IF (TRIG_valve_tank_R.Q	OR Timer_valveQ = TRUE) THEN
	HW_valve_pomp_teplica :=	FALSE;
	Timer_valveQ	:= FALSE;
	Timer_valve.IN	:= FALSE;
END_IF



IF (TRIG_start_poliv.Q AND  Modbus.Teplica_poliv_status_PLC <> 2)   THEN
		Cnt_cleared	:= 	FALSE;
		Step_1_clear	 :=	FALSE;
		Poliv_liters	:=	0;
		FertA_liters	:=	0;
		FertB_liters	:=	0;
		Cnt_water_fertA_start	:=	0;
		Cnt_water_fertB_start	:=	0;
		Modbus.Cnt_water_fertA	:=	0;
		Modbus.Cnt_water_fertB	:=	0;
		Modbus.Teplica_DI1_poliv	:=	0;
		Modbus.Teplica_DI2_fertA	:=	0;
		Modbus.Teplica_DI3_fertB	:=	0;
		Modbus.Teplica_poliv_status_PLC:=1;
		Modbus.Teplica_poliv_message_PLC:=1;
		Modbus.Teplica_time_elapsed_poliv :=0;
		Modbus.Teplica_time_elapsed_fertA :=0;
		Modbus.Teplica_time_elapsed_fertB :=0;

		Timer_1_clearQ			:= FALSE;
		Timer_2_fertAQ			:= FALSE;
		Timer_3_clearQ			:= FALSE;
		Timer_4_fertBQ			:= FALSE;
		Step_1_clear				:= FALSE;
		Poliv_init_stop			:= FALSE;
		FertA_init_stop			:=	FALSE;
		FertB_init_stop			:=	FALSE;
		Bool_poliv_before_fert		:=	FALSE;
END_IF

(*ограничитель полива  в случае невозможности обнулить счётчики из-за недоступности RS485-шлюза*)
(*
	IF (Poliv_init_stop	=	FALSE AND (Modbus.Teplica_poliv_break=TRUE  OR  Cnt_Teplica_poliv_message_PLC_M3 > 2 OR  Cnt_Teplica_poliv_message_PLC_M5 > 2 OR  Cnt_Teplica_poliv_message_PLC_M7 > 2 OR  Cnt_Teplica_poliv_message_PLC_M9 > 2 OR  Cnt_Teplica_poliv_message_PLC_M11 > 2))
	THEN
		Cnt_cleared	:= 	FALSE;
		Modbus.Teplica_poliv_status_PLC :=  0;
		Poliv_init_stop	:=	TRUE;
		Modbus.Teplica_poliv_active:= FALSE;

		Modbus.Teplica_DO4_pomp_poliv:=FALSE;
		Modbus.Teplica_DO5_pomp_fertA :=  FALSE;
		Modbus.Teplica_DO6_pomp_fertB :=  FALSE;

		Step_1_clear	 :=	FALSE;

		Timer_poliv_all.IN := FALSE;
		Timer_1_clear.IN := FALSE;
		Timer_2_fertA.IN:=FALSE;
		Timer_3_clear.IN := FALSE;
		Timer_4_fertB.IN:=FALSE;
	END_IF
*)

(*Нормальный режим старта полива после обнуления счётчиков*)

IF (Modbus.Teplica_poliv_status_PLC=2 AND Cnt_cleared=TRUE AND Step_1_clear = FALSE ) THEN
	DO3_poliv_writed_0		:=	FALSE;
	DO4_fertA_writed_0		:=	FALSE;
	DO5_fertB_writed_0		:=	FALSE;

	Step_1_clear	 :=	TRUE;
	Modbus.Teplica_DO4_pomp_poliv:=TRUE;
	 t_Started_poliv := TIME();
	Timer_poliv_all(IN:=NOT Timer_poliv_allQ , PT:=tTimerValue_poliv_all , Q=>Timer_poliv_allQ , ET=> );
	Timer_poliv_with_fert(IN:=NOT Timer_poliv_with_fertQ , PT:=tTimerValue_poliv_with_fert , Q=>Timer_poliv_with_fertQ , ET=> );
	Timer_1_clear(IN:=NOT Timer_1_clearQ , PT:=tTimerValue_1_clear , Q=>Timer_1_clearQ , ET=> );
END_IF

IF (Modbus.Teplica_poliv_status_PLC=2 AND Cnt_cleared=TRUE  ) THEN


	Poliv_liters 	:= 	UDINT_TO_REAL(Modbus.Teplica_DI1_poliv)/INT_TO_REAL(Modbus.Teplica_poliv_kf);
	FertA_liters	:=	UDINT_TO_REAL(Modbus.Teplica_DI2_fertA)/INT_TO_REAL(Modbus.Teplica_fertA_kf);
	FertB_liters	:=	UDINT_TO_REAL(Modbus.Teplica_DI3_fertB)/INT_TO_REAL(Modbus.Teplica_fertB_kf);
	Modbus.Teplica_time_elapsed_poliv :=(TIME_TO_UDINT( TIME() - t_Started_poliv))/1000;

(* промывка и фертигация   OR Modbus.Teplica_set_poliv_before_fert >Poliv_liters*)

IF (Modbus.Teplica_type_poliv = TRUE) THEN
	IF ((Timer_1_clear.Q OR Poliv_liters>Modbus.Teplica_set_poliv_before_fert) AND Bool_poliv_before_fert=FALSE) THEN
		Timer_1_clear.IN 		:= FALSE;
		Bool_poliv_before_fert	:= TRUE;
		IF (Modbus.Teplica_type_fert = FALSE) THEN
			Modbus.Teplica_DO5_pomp_fertA :=  TRUE;  (*включение насоса фертигации из бака А*)
			Timer_2_fertA(IN:=NOT Timer_2_fertAQ , PT:=tTimerValue_2_fertA , Q=>Timer_2_fertAQ , ET=> );
			t_Started_fertA := TIME();
			Cnt_water_fertA_start :=Modbus.Teplica_DI1_poliv;


		ELSE
			Modbus.Teplica_DO6_pomp_fertB :=  TRUE;   (*включение насоса фертигации из бака B*)
			Timer_4_fertB(IN:=NOT Timer_4_fertBQ , PT:=tTimerValue_4_fertB , Q=>Timer_4_fertBQ , ET=> );
			t_Started_fertB := TIME();
			Cnt_water_fertB_start :=Modbus.Teplica_DI1_poliv;

		END_IF


	END_IF





	IF ( (Timer_2_fertA.Q OR FertA_liters > Modbus.Teplica_set_fertA) AND Modbus.Teplica_DO5_pomp_fertA =  TRUE) THEN
		Modbus.Teplica_DO5_pomp_fertA :=  FALSE; (*отключение насоса фертигации из бака А*)
		Timer_2_fertA.IN:=FALSE;
		FertA_init_stop	:=	TRUE;
		Timer_3_clear(IN:=NOT Timer_3_clearQ , PT:=tTimerValue_3_clear , Q=>Timer_3_clearQ , ET=> );
	END_IF

	IF ( (Timer_4_fertB.Q OR FertB_liters > Modbus.Teplica_set_fertB) AND Modbus.Teplica_DO6_pomp_fertB =  TRUE ) THEN
		Modbus.Teplica_DO6_pomp_fertB :=  FALSE; (*отключение насоса фертигации из бака B*)
		Timer_4_fertB.IN:=FALSE;
		FertB_init_stop	:=	TRUE;
		Timer_3_clear(IN:=NOT Timer_3_clearQ , PT:=tTimerValue_3_clear , Q=>Timer_3_clearQ , ET=> );
	END_IF

END_IF

(*ограничитель полива  в нормальном режиме*)
	IF (Modbus.Teplica_type_poliv = FALSE) THEN
		IF ((Timer_poliv_all.Q=TRUE OR (Poliv_liters > Modbus.Teplica_set_poliv)  OR Modbus.Teplica_poliv_break=TRUE OR Timer_3_clear.Q=TRUE) AND  Poliv_init_stop = FALSE )THEN
			IF (Modbus.Teplica_DO5_pomp_fertA =  TRUE) THEN
				Modbus.Teplica_time_elapsed_fertA :=(TIME_TO_UDINT( TIME() - t_Started_fertA))/1000;
			END_IF
			IF (Modbus.Teplica_DO6_pomp_fertB =  TRUE) THEN
				Modbus.Teplica_time_elapsed_fertB :=(TIME_TO_UDINT( TIME() - t_Started_fertB))/1000;
			END_IF

			Poliv_init_stop	:=	TRUE;
			Cnt_cleared	:= 	FALSE;
			Modbus.Teplica_poliv_status_PLC :=  0;
			Modbus.Teplica_poliv_active:= FALSE;
			Modbus.Teplica_DO4_pomp_poliv:=FALSE;
			Modbus.Teplica_DO5_pomp_fertA :=  FALSE;
			Modbus.Teplica_DO6_pomp_fertB :=  FALSE;
			Timer_poliv_all.IN := FALSE;
			Timer_poliv_with_fert.IN := FALSE;
			Timer_1_clear.IN := FALSE;
			Timer_2_fertA.IN:=FALSE;
			Timer_3_clear.IN := FALSE;
			Timer_4_fertB.IN:=FALSE;
		END_IF
	ELSE
		IF ((Timer_poliv_with_fert.Q=TRUE OR   Modbus.Teplica_poliv_break=TRUE OR Timer_3_clear.Q=TRUE) AND  Poliv_init_stop = FALSE )THEN
			IF (Modbus.Teplica_DO5_pomp_fertA =  TRUE) THEN
				Modbus.Teplica_time_elapsed_fertA :=(TIME_TO_UDINT( TIME() - t_Started_fertA))/1000;
			END_IF
			IF (Modbus.Teplica_DO6_pomp_fertB =  TRUE) THEN
				Modbus.Teplica_time_elapsed_fertB :=(TIME_TO_UDINT( TIME() - t_Started_fertB))/1000;
			END_IF

			Poliv_init_stop	:=	TRUE;
			Cnt_cleared	:= 	FALSE;
			Modbus.Teplica_poliv_status_PLC :=  0;
			Modbus.Teplica_poliv_active:= FALSE;
			Modbus.Teplica_DO4_pomp_poliv:=FALSE;
			Modbus.Teplica_DO5_pomp_fertA :=  FALSE;
			Modbus.Teplica_DO6_pomp_fertB :=  FALSE;
			Timer_poliv_all.IN := FALSE;
			Timer_poliv_with_fert.IN := FALSE;
			Timer_1_clear.IN := FALSE;
			Timer_2_fertA.IN:=FALSE;
			Timer_3_clear.IN := FALSE;
			Timer_4_fertB.IN:=FALSE;
		END_IF
	END_IF
END_IF











(*LIGHT TEPLICA *)

IF (Modbus.Teplica_DO3_light = FALSE) THEN

	IF ((Modbus.Teplica_light_lux > Modbus.Teplica_light_set_low+gisterezis_lux) OR Modbus.Teplica_light_allow = FALSE  ) THEN
		Modbus.Teplica_DO3_light :=FALSE;
	END_IF

	IF ((Modbus.Teplica_light_lux <  Modbus.Teplica_light_set_low-gisterezis_lux ) AND Modbus.Teplica_light_allow ) THEN
		Modbus.Teplica_DO3_light:=TRUE;
	END_IF

END_IF

IF (Modbus.Teplica_DO3_light = TRUE) THEN

	IF ((Modbus.Teplica_light_lux-Modbus.Teplica_power_light_lux > Modbus.Teplica_light_set_low+gisterezis_lux) OR Modbus.Teplica_light_allow = FALSE  ) THEN
		Modbus.Teplica_DO3_light :=FALSE;
	END_IF

	IF ((Modbus.Teplica_light_lux-Modbus.Teplica_power_light_lux <  Modbus.Teplica_light_set_low-gisterezis_lux ) AND Modbus.Teplica_light_allow ) THEN
		Modbus.Teplica_DO3_light:=TRUE;
	END_IF

END_IF



(*HEAT TEPLICA *)

	IF ((Modbus.Teplica_temp_air > Modbus.Teplica_temp_set_low+1)   ) THEN
		Modbus.Teplica_DO2_heat :=FALSE;
	END_IF

	IF ((Modbus.Teplica_temp_air <  Modbus.Teplica_temp_set_low-1 ) ) THEN
		Modbus.Teplica_DO2_heat:=TRUE;
	END_IF

(*VENT  TEPLICA *)

	IF ((Modbus.Teplica_temp_air < Modbus.Teplica_temp_set_high-1)   ) THEN
		Modbus.Teplica_DO1_vent			 :=FALSE;
	END_IF

	IF ((Modbus.Teplica_temp_air >  Modbus.Teplica_temp_set_high+1 ) ) THEN
		Modbus.Teplica_DO1_vent:=TRUE;
	END_IF


	IF (Modbus.Teplica_temp_air < Modbus.Teplica_set_temp_window_open-1 ) THEN
		HW_window_opener				:=FALSE;
		Modbus.Teplica_window_opener	:=FALSE;
	END_IF
	IF (Modbus.Teplica_temp_air >  Modbus.Teplica_set_temp_window_open+1 AND   Modbus.Street_temp > 5 ) THEN
		HW_window_opener				:=TRUE;
		Modbus.Teplica_window_opener	:=TRUE;
	END_IF


	IF (Modbus.Teplica_temp_air < Modbus.Teplica_set_temp_pomp_cold-2   ) THEN
		HW_pomp_cold				:=FALSE;
		Modbus.Teplica_pomp_cold	:=FALSE;
	END_IF
	IF (Modbus.Teplica_temp_air >  Modbus.Teplica_set_temp_pomp_cold+2 AND   Modbus.Street_temp > 5 ) THEN
		HW_pomp_cold				:=TRUE;
		Modbus.Teplica_pomp_cold	:=TRUE;
	END_IF
END_PROGRAM

(* POU teplica_ai, ST *)
PROGRAM teplica_ai
VAR
    (* Общие таймеры *)
    Timer_poliv_all : TON;
    Timer_poliv_with_fert : TON;
    Timer_1_clear : TON;
    Timer_3_clear : TON;
    Timer_poliv_finish : TON;
    Timer_calc_kf : TON;
    Timer_valve : TON;

    (* Таймеры для баков (A и B) *)
    Timer_fert : ARRAY[1..2] OF TON;
    Timer_fertQ : ARRAY[1..2] OF BOOL;

    (* Триггеры *)
    TRIG_start_poliv : R_TRIG;
    TRIG_poliv_break : R_TRIG;
    TRIG_valve_tank_F : F_TRIG;
    TRIG_valve_tank_R : R_TRIG;
    TRIG_level_tank_low : R_TRIG;
    TRIG_level_tank_high : R_TRIG;

    (* ПИ-регуляторы и их параметры (для двух баков) *)
    pi_fert : ARRAY[1..2] OF FB_CTRL_PI;
    pi_par : ARRAY[1..2] OF ST_CTRL_PI_PARAMS;
    kf_calc : ARRAY[1..2] OF REAL;
    cnt_water_fert_start : ARRAY[1..2] OF UDINT;
    cnt_fert_calc_start : ARRAY[1..2] OF REAL;
    vol_fert : ARRAY[1..2] OF REAL;
    fOut : ARRAY[1..2] OF REAL;
    act : ARRAY[1..2] OF REAL;
    pwm_data : ARRAY[1..2] OF REAL;
    pwm_cnt : ARRAY[1..2] OF UDINT;
    pwm_avg : ARRAY[1..2] OF REAL;
    fert_pwm_level : ARRAY[1..2] OF UINT;

    (* Переменные для объёмов *)
    Poliv_liters : REAL;
    FertA_liters : REAL;
    FertB_liters : REAL;
    Cnt_water_calc_kf_start : REAL;
    vol_water : REAL;

    (* Прочие переменные *)
    Cnt_water_pipe : UDINT;
    Cnt_water_finish_clear_start : UDINT;
    Cnt_water_finish_clear : REAL;
    t_Started_poliv : TIME;
    t_Started_fert : ARRAY[1..2] OF TIME;
    tTimerValue_poliv_all : TIME := t#60s;
    tTimerValue_1_clear : TIME := t#10s;
    tTimerValue_2_fert : ARRAY[1..2] OF TIME := t#30s, t#10s;
    tTimerValue_3_clear : TIME := t#60s;
    tTimerValue_poliv_with_fert : TIME := t#60m;
    tTimerValue_poliv_finish : TIME := t#3s;
    tTimerValue_valve_water : TIME := t#60m;
    Bool_poliv_before_fert : BOOL;
    max_EC : REAL;
    avg_light_ma : FB_CTRL_MOVING_AVERAGE;
    stParams_avg_light : ST_CTRL_MOVING_AVERAGE_PARAMS;
    arr_table : ARRAY[1..20] OF FLOAT;
    start_cfg_avg_light : BOOL;
    start_cfg_pi_par : BOOL;
    gisterezis_lux : INT := 1000;
    tank_level_low : BOOL;
    tank_level_high : BOOL;
    fert_idx : INT;
    setpoint : REAL;
    zone_offset : INT;
END_VAR
(* ---------- Инициализация скользящего среднего ---------- *)
IF NOT start_cfg_avg_light THEN
    stParams_avg_light.tCtrlCycleTime := T#60s;
    stParams_avg_light.tTaskCycleTime := T#10ms;
    stParams_avg_light.nSamplesToFilter := 20;
    stParams_avg_light.pWorkArray_ADR := ADR(arr_table);
    stParams_avg_light.nWorkArray_SIZEOF := SIZEOF(arr_table);
    start_cfg_avg_light := TRUE;
END_IF
avg_light_ma(fIn:=Modbus.Teplica_light_lux, fManSyncValue:=0, bSync:=0,
             eMode:=eCTRL_MODE_ACTIVE, bHold:=0, stParams:=stParams_avg_light,
             fOut=>Modbus.Teplica_avg_lux);

(* ---------- Инициализация ПИ-регуляторов и коэффициентов ---------- *)
IF NOT start_cfg_pi_par THEN
    FOR fert_idx := 1 TO 2 DO
        pi_par[fert_idx].bARWOnIPartOnly := 0;
        pi_par[fert_idx].fKp := 300000;
        pi_par[fert_idx].fOutMaxLimit := 32765;
        pi_par[fert_idx].fOutMinLimit := 16800;
        pi_par[fert_idx].tCtrlCycleTime := T#4s;
        pi_par[fert_idx].tTaskCycleTime := T#10ms;
        pi_par[fert_idx].tTn := T#8s;
        kf_calc[fert_idx] := 12.0;   (* начальное значение Kf *)
    END_FOR
    start_cfg_pi_par := TRUE;
END_IF

(* ---------- Защита от нулевых коэффициентов ---------- *)
FOR fert_idx := 1 TO 2 DO
    IF kf_calc[fert_idx] = 0.0 THEN
        kf_calc[fert_idx] := 12.0;
    END_IF
END_FOR
IF Modbus.Teplica_fert_kf = 0 THEN
    Modbus.Teplica_fert_kf := 24;
END_IF
setpoint := 1.0 / INT_TO_REAL(Modbus.Teplica_fert_kf);

(* ---------- Установка времён из Modbus (перевод минут в мс) ---------- *)
tTimerValue_poliv_all        := UDINT_TO_TIME(60000 * Modbus.Teplica_set_max_poliv_time);
tTimerValue_1_clear          := UDINT_TO_TIME(60000 * Modbus.Teplica_set_clear_time);
tTimerValue_2_fert[1]        := UDINT_TO_TIME(60000 * Modbus.Teplica_set_max_fertA_time);
tTimerValue_2_fert[2]        := UDINT_TO_TIME(60000 * Modbus.Teplica_set_max_fertB_time);
tTimerValue_3_clear          := UDINT_TO_TIME(60000 * Modbus.Teplica_set_finish_clear_time);

(* ---------- Вызов таймеров ---------- *)
Timer_poliv_all();
Timer_poliv_with_fert();
Timer_1_clear();
Timer_3_clear();
FOR fert_idx := 1 TO 2 DO Timer_fert[fert_idx](); END_FOR
Timer_poliv_finish();
Timer_calc_kf();
Timer_valve();

(* ---------- Триггеры ---------- *)
TRIG_start_poliv(CLK := Modbus.Teplica_poliv_active);
TRIG_poliv_break(CLK := Modbus.Teplica_poliv_break);
TRIG_valve_tank_F(CLK := HW_water_tank_teplica_level);
TRIG_valve_tank_R(CLK := HW_water_tank_teplica_level);

tank_level_low   := Modbus.Teplica_tank_level < 1000;
tank_level_high  := Modbus.Teplica_tank_level > 1200;
TRIG_level_tank_low(CLK := tank_level_low);
TRIG_level_tank_high(CLK := tank_level_high);
Modbus.Teplica_tank_teplica_level := HW_water_tank_teplica_level;

(* ---------- Управление клапаном воды в бак ---------- *)
IF TRIG_valve_tank_F.Q OR TRIG_level_tank_low.Q THEN
    Timer_valve(IN := NOT Timer_valve.Q, PT := tTimerValue_valve_water);
    HW_valve_pomp_teplica := TRUE;
    Modbus.Teplica_valve_water_in := TRUE;
END_IF
IF TRIG_valve_tank_R.Q OR Timer_valve.Q OR TRIG_level_tank_high.Q THEN
    HW_valve_pomp_teplica := FALSE;
    Modbus.Teplica_valve_water_in := FALSE;
    Timer_valve.IN := FALSE;
END_IF

(* ---------- Старт полива ---------- *)
IF TRIG_start_poliv.Q AND Modbus.Teplica_tank_level > 400 THEN
    FOR fert_idx := 1 TO 2 DO
        pwm_data[fert_idx] := 0.0;
        pwm_cnt[fert_idx] := 0;
        pwm_avg[fert_idx] := 0.0;
        cnt_water_fert_start[fert_idx] := 0;
        cnt_fert_calc_start[fert_idx] := 0.0;
    END_FOR
    Modbus.Teplica_impulse_fertA_cnt := 0;
    Modbus.Teplica_impulse_fertB_cnt := 0;
    Modbus.Teplica_impulse_water_cnt := 0;
    Modbus.Teplica_cnt_water_pipe := 0;
    Modbus.Teplica_time_elapsed_poliv := 0;
    Modbus.Teplica_time_elapsed_fertA := 0;
    Modbus.Teplica_time_elapsed_fertB := 0;
    Poliv_liters := 0.0;
    FertA_liters := 0.0;
    FertB_liters := 0.0;
    Cnt_water_finish_clear := 0.0;
    Cnt_water_finish_clear_start := 0;
    Cnt_water_calc_kf_start := 0.0;
    max_EC := 0.0;
    Bool_poliv_before_fert := FALSE;

    FOR fert_idx := 1 TO 2 DO
        Timer_fert[fert_idx].IN := FALSE;
    END_FOR
    Timer_1_clear.IN := FALSE;
    Timer_3_clear.IN := FALSE;
    Timer_calc_kf.IN := FALSE;
    Timer_poliv_finish.IN := FALSE;
    Timer_poliv_all.IN := FALSE;
    Timer_poliv_with_fert.IN := FALSE;

    Modbus.Teplica_pomp_poliv := TRUE;
    t_Started_poliv := TIME();
    Timer_poliv_all(IN := NOT Timer_poliv_all.Q, PT := tTimerValue_poliv_all);
    Timer_poliv_with_fert(IN := NOT Timer_poliv_with_fert.Q, PT := tTimerValue_poliv_with_fert);
    Timer_1_clear(IN := NOT Timer_1_clear.Q, PT := tTimerValue_1_clear);
    Modbus.Teplica_poliv_status_PLC := 2;
    (* вычисляем смещение для зоны *)
    zone_offset := 0;
    IF Modbus.Teplica_zone_poliv <> 0 THEN zone_offset := 1; END_IF
    Modbus.Teplica_poliv_message_PLC := 1 + zone_offset;
END_IF

(* ---------- Основной цикл полива ---------- *)
IF Modbus.Teplica_poliv_status_PLC = 2 THEN
    Cnt_water_pipe := Modbus.Teplica_cnt_water_pipe;
    Poliv_liters  := UDINT_TO_REAL(Modbus.Teplica_impulse_water_cnt) / INT_TO_REAL(Modbus.Teplica_poliv_kf);
    FertA_liters  := UDINT_TO_REAL(Modbus.Teplica_impulse_fertA_cnt) / INT_TO_REAL(Modbus.Teplica_fertA_kf);
    FertB_liters  := UDINT_TO_REAL(Modbus.Teplica_impulse_fertB_cnt) / INT_TO_REAL(Modbus.Teplica_fertB_kf);
    Modbus.Teplica_time_elapsed_poliv := (TIME_TO_UDINT(TIME() - t_Started_poliv)) / 1000;
    IF Modbus.Teplica_sensor_soil_EC > max_EC THEN max_EC := Modbus.Teplica_sensor_soil_EC; END_IF

    (* выбор бака: 1 – A, 2 – B *)
    IF Modbus.Teplica_type_fert THEN
        fert_idx := 2;
    ELSE
        fert_idx := 1;
    END_IF

    (* смещение для зоны (используется далее) *)
    zone_offset := 0;
    IF Modbus.Teplica_zone_poliv <> 0 THEN zone_offset := 1; END_IF

    (* ------------------- Полив с фертигацией ------------------- *)
    IF Modbus.Teplica_type_poliv THEN
        (* Этап 1: промывка перед фертигацией *)
        IF NOT Timer_1_clear.Q AND NOT Bool_poliv_before_fert THEN
            Modbus.Teplica_poliv_message_PLC := 3 + (fert_idx-1)*2 + zone_offset;
        END_IF

        (* Переход к фертигации *)
        IF (Timer_1_clear.Q OR Poliv_liters > Modbus.Teplica_set_poliv_before_fert) AND NOT Bool_poliv_before_fert THEN
            Timer_1_clear.IN := FALSE;
            Bool_poliv_before_fert := TRUE;
            IF fert_idx = 1 THEN
                Modbus.Teplica_pomp_fertA := TRUE;
            ELSE
                Modbus.Teplica_pomp_fertB := TRUE;
            END_IF
            Timer_fert[fert_idx](IN := NOT Timer_fert[fert_idx].Q, PT := tTimerValue_2_fert[fert_idx]);
            t_Started_fert[fert_idx] := TIME();
            cnt_water_fert_start[fert_idx] := Modbus.Teplica_impulse_water_cnt;
            cnt_fert_calc_start[fert_idx] := Poliv_liters;
            Cnt_water_calc_kf_start := Poliv_liters;
            Modbus.Teplica_poliv_message_PLC := 7 + (fert_idx-1)*2 + zone_offset;
        END_IF

        (* Работа активного бака *)
        IF (fert_idx = 1 AND Modbus.Teplica_pomp_fertA) OR (fert_idx = 2 AND Modbus.Teplica_pomp_fertB) THEN
            act[fert_idx] := 1.0 / kf_calc[fert_idx];
            pi_fert[fert_idx](fSetpointValue := setpoint, fActualValue := act[fert_idx],
                fManSyncValue := 0, bSync := 0, eMode := 2, bHold := 0,
                stParams := pi_par[fert_idx], fOut => fOut[fert_idx]);

            IF fert_idx = 1 THEN
                Modbus.Teplica_time_elapsed_fertA := (TIME_TO_UDINT(TIME() - t_Started_fert[1])) / 1000;
                Modbus.Cnt_water_fertA := Modbus.Teplica_impulse_water_cnt - cnt_water_fert_start[1];
            ELSE
                Modbus.Teplica_time_elapsed_fertB := (TIME_TO_UDINT(TIME() - t_Started_fert[2])) / 1000;
                Modbus.Cnt_water_fertB := Modbus.Teplica_impulse_water_cnt - cnt_water_fert_start[2];
            END_IF

            Timer_calc_kf(IN := NOT Timer_calc_kf.Q, PT := t#3s);
            IF Timer_calc_kf.Q THEN
                vol_water := Poliv_liters - Cnt_water_calc_kf_start;
                IF fert_idx = 1 THEN
                    vol_fert[1] := FertA_liters - cnt_fert_calc_start[1];
                ELSE
                    vol_fert[2] := FertB_liters - cnt_fert_calc_start[2];
                END_IF
                IF vol_fert[fert_idx] > 0.0 THEN
                    kf_calc[fert_idx] := vol_water / vol_fert[fert_idx];
                ELSE
                    kf_calc[fert_idx] := 1000.0;
                END_IF
                Cnt_water_calc_kf_start := Poliv_liters;
                IF fert_idx = 1 THEN
                    cnt_fert_calc_start[1] := FertA_liters;
                ELSE
                    cnt_fert_calc_start[2] := FertB_liters;
                END_IF
                Timer_calc_kf.IN := FALSE;
            END_IF

            fert_pwm_level[fert_idx] := REAL_TO_UINT(fOut[fert_idx]);
            pwm_data[fert_idx] := pwm_data[fert_idx] + fert_pwm_level[fert_idx];
            pwm_cnt[fert_idx] := pwm_cnt[fert_idx] + 1;
            pwm_avg[fert_idx] := pwm_data[fert_idx] / pwm_cnt[fert_idx];
        END_IF

        (* Завершение фертигации (переход к промывке) *)
        IF (fert_idx = 1 AND Modbus.Teplica_pomp_fertA) AND (Timer_fert[1].Q OR FertA_liters > Modbus.Teplica_set_fertA) THEN
            Modbus.Teplica_pomp_fertA := FALSE;
            Modbus.Teplica_time_elapsed_fertA := (TIME_TO_UDINT(TIME() - t_Started_fert[1])) / 1000;
            Modbus.Cnt_water_fertA := Modbus.Teplica_impulse_water_cnt - cnt_water_fert_start[1];
            Timer_fert[1].IN := FALSE;
            Cnt_water_finish_clear_start := Modbus.Teplica_impulse_water_cnt;
            Timer_3_clear(IN := NOT Timer_3_clear.Q, PT := tTimerValue_3_clear);
            Modbus.Teplica_poliv_message_PLC := 11 + zone_offset;
        END_IF
        IF (fert_idx = 2 AND Modbus.Teplica_pomp_fertB) AND (Timer_fert[2].Q OR FertB_liters > Modbus.Teplica_set_fertB) THEN
            Modbus.Teplica_pomp_fertB := FALSE;
            Modbus.Teplica_time_elapsed_fertB := (TIME_TO_UDINT(TIME() - t_Started_fert[2])) / 1000;
            Modbus.Cnt_water_fertB := Modbus.Teplica_impulse_water_cnt - cnt_water_fert_start[2];
            Timer_fert[2].IN := FALSE;
            Cnt_water_finish_clear_start := Modbus.Teplica_impulse_water_cnt;
            Timer_3_clear(IN := NOT Timer_3_clear.Q, PT := tTimerValue_3_clear);
            Modbus.Teplica_poliv_message_PLC := 13 + zone_offset;
        END_IF

        (* Расчёт объёма промывки *)
        IF Modbus.Teplica_poliv_message_PLC >= 11 AND Modbus.Teplica_poliv_message_PLC <= 14 THEN
            Cnt_water_finish_clear := UDINT_TO_REAL(Modbus.Teplica_impulse_water_cnt - Cnt_water_finish_clear_start) / Modbus.Teplica_poliv_kf;
        END_IF

        (* Условия окончания полива с фертигацией *)
        IF Timer_poliv_with_fert.Q OR Modbus.Teplica_poliv_break OR Timer_3_clear.Q OR
           Cnt_water_finish_clear > Modbus.Teplica_set_finish_clear_vol THEN
            Modbus.Teplica_max_EC := max_EC;
            Modbus.Teplica_poliv_active := FALSE;
            Modbus.Teplica_pomp_poliv := FALSE;
            Modbus.Teplica_pomp_fertA := FALSE;
            Modbus.Teplica_pomp_fertB := FALSE;
            Timer_poliv_all.IN := FALSE;
            Timer_poliv_with_fert.IN := FALSE;
            Timer_1_clear.IN := FALSE;
            Timer_3_clear.IN := FALSE;
            FOR fert_idx := 1 TO 2 DO
                Timer_fert[fert_idx].IN := FALSE;
            END_FOR
            Timer_calc_kf.IN := FALSE;
            Modbus.Teplica_poliv_message_PLC := 15 + (fert_idx-1)*2 + zone_offset;
            Modbus.Teplica_poliv_status_PLC := 10;
            Timer_poliv_finish(IN := NOT Timer_poliv_finish.Q, PT := tTimerValue_poliv_finish);
        END_IF

    (* ------------------- Полив без фертигации ------------------- *)
    ELSE
        IF Timer_poliv_all.Q OR (Poliv_liters > Modbus.Teplica_set_poliv) OR Modbus.Teplica_poliv_break THEN
            Modbus.Teplica_poliv_message_PLC := 19 + zone_offset;
            Modbus.Teplica_poliv_active := FALSE;
            Modbus.Teplica_pomp_poliv := FALSE;
            Modbus.Teplica_pomp_fertA := FALSE;
            Modbus.Teplica_pomp_fertB := FALSE;
            Timer_poliv_all.IN := FALSE;
            Timer_poliv_with_fert.IN := FALSE;
            Timer_1_clear.IN := FALSE;
            Timer_3_clear.IN := FALSE;
            FOR fert_idx := 1 TO 2 DO
                Timer_fert[fert_idx].IN := FALSE;
            END_FOR
            Modbus.Teplica_poliv_status_PLC := 10;
        END_IF
    END_IF

    (* Обнуление ШИМ, если насосы не активны *)
    IF NOT Modbus.Teplica_type_poliv OR (Modbus.Teplica_type_poliv AND NOT (Modbus.Teplica_pomp_fertA OR Modbus.Teplica_pomp_fertB)) THEN
        fert_pwm_level[1] := 0;
        fert_pwm_level[2] := 0;
    END_IF

    (* Вывод данных для Modbus *)
    Modbus.Teplica_fert_actA := kf_calc[1];
    Modbus.Teplica_fert_actB := kf_calc[2];
    Modbus.Teplica_fert_pwm_levelA := REAL_TO_INT(100.0 * fert_pwm_level[1] / 32765.0);
    Modbus.Teplica_fert_pwm_levelB := REAL_TO_INT(100.0 * fert_pwm_level[2] / 32765.0);
    Modbus.Teplica_pwm_avg_A := REAL_TO_INT(100.0 * pwm_avg[1] / 32765.0);
    Modbus.Teplica_pwm_avg_B := REAL_TO_INT(100.0 * pwm_avg[2] / 32765.0);
END_IF

(* ---------- Управление освещением ---------- *)
IF Modbus.Teplica_light THEN
    IF (Modbus.Teplica_avg_lux > Modbus.Teplica_light_set_low + gisterezis_lux) OR (Modbus.Teplica_temp_air > 28) OR NOT Modbus.Teplica_light_allow THEN
        Modbus.Teplica_light := FALSE;
        HW_teplica_light := FALSE;
    END_IF
ELSE
    IF (Modbus.Teplica_avg_lux < Modbus.Teplica_light_set_low - gisterezis_lux) AND (Modbus.Teplica_temp_air < 27) AND Modbus.Teplica_light_allow THEN
        Modbus.Teplica_light := TRUE;
        HW_teplica_light := TRUE;
    END_IF
END_IF

(* ---------- Управление отоплением ---------- *)
IF Modbus.Teplica_temp_air > Modbus.Teplica_temp_set_low + 1 THEN
    Modbus.Teplica_heat := FALSE;
    HW_teplica_heat := FALSE;
ELSIF Modbus.Teplica_temp_air < Modbus.Teplica_temp_set_low - 1 THEN
    Modbus.Teplica_heat := TRUE;
    HW_teplica_heat := TRUE;
END_IF

(* ---------- Управление подогревом бака ---------- *)
IF (Modbus.Teplica_temp_water_tank > Modbus.Teplica_set_temp_tank + 1) OR HW_teplica_heat OR (Modbus.Teplica_tank_level < 400) THEN
    Modbus.Teplica_tank_heat := FALSE;
    HW_teplica_tank_heat := FALSE;
ELSIF (Modbus.Teplica_temp_water_tank < Modbus.Teplica_set_temp_tank - 1) AND NOT HW_teplica_heat AND (Modbus.Teplica_tank_level > 400) THEN
    Modbus.Teplica_tank_heat := TRUE;
    HW_teplica_tank_heat := TRUE;
END_IF

(* ---------- Управление вентиляцией ---------- *)
IF Modbus.Teplica_temp_air < Modbus.Teplica_temp_set_high - 1 THEN
    Modbus.Teplica_vent := FALSE;
    HW_teplica_vent := FALSE;
ELSIF Modbus.Teplica_temp_air > Modbus.Teplica_temp_set_high + 1 THEN
    Modbus.Teplica_vent := TRUE;
    HW_teplica_vent := TRUE;
END_IF

(* ---------- Открытие форточки ---------- *)
IF Modbus.Teplica_temp_air < Modbus.Teplica_set_temp_window_open - 1 THEN
    HW_teplica_window_opener := FALSE;
    Modbus.Teplica_window_opener := FALSE;
ELSIF Modbus.Teplica_temp_air > Modbus.Teplica_set_temp_window_open + 1 AND Modbus.Street_temp > 0 THEN
    HW_teplica_window_opener := TRUE;
    Modbus.Teplica_window_opener := TRUE;
END_IF

(* ---------- Холодный насос ---------- *)
IF Modbus.Teplica_temp_air < Modbus.Teplica_set_temp_pomp_cold - 1 THEN
    HW_teplica_pomp_cold := FALSE;
    Modbus.Teplica_pomp_cold := FALSE;
ELSIF Modbus.Teplica_temp_air > Modbus.Teplica_set_temp_pomp_cold + 1 AND Modbus.Street_temp > 10 THEN
    HW_teplica_pomp_cold := TRUE;
    Modbus.Teplica_pomp_cold := TRUE;
END_IF
END_PROGRAM

(* POU teplica_new_2025, ST *)
PROGRAM teplica_new_2025
VAR
	Cnt_water_fertA_start	:	UDINT;
	Cnt_water_fertB_start	:	UDINT;
	Cnt_water_finish_clear_start	:	UDINT;
	Cnt_water_finish_clear	:		REAL;
	t_Started_poliv			:	TIME;
	t_Started_fertA			:	TIME;
	t_Started_fertB			:	TIME;


	Timer_poliv_all			: TON;
	Timer_poliv_allQ			: BOOL;

	Timer_1_clear			: TON;
	Timer_2_fertA				: TON;
	Timer_3_clear			: TON;
	Timer_4_fertB				: TON;
	Timer_poliv_with_fert		: TON;
	Timer_poliv_finish			: TON;

	Timer_calc_kf			: TON;
	Timer_calc_kfQ			:BOOL;
	Cnt_water_calc_kf_start		:REAL;
	Cnt_fertA_calc_kf_start		:REAL;
	Cnt_fertB_calc_kf_start		:REAL;
	Kf_calc_fertA				: REAL:=12;
	Kf_calc_fertB				: REAL:=12;
	vol_water				: REAL;
	vol_fertA					: REAL;
	vol_fertB					: REAL;

	Timer_poliv_finishQ		: BOOL;
	Timer_1_clearQ			: BOOL;
	Timer_2_fertAQ			: BOOL;
	Timer_3_clearQ			: BOOL;
	Timer_4_fertBQ			: BOOL;



	 tTimerValue_poliv_all		: TIME:=t#60s;  (* Максимальное время полива*)
	 tTimerValue_1_clear		: TIME:=t#10s;  (* Промывка перед 1 фертигацией*)
	 tTimerValue_2_fertA		: TIME:=t#30s;  (* Ограничение фертигации из бака А*)
	 tTimerValue_3_clear		: TIME:=t#60s;  (* Промывка перед OFF*)
	 tTimerValue_4_fertB		: TIME:=t#10s;  (* Ограничение фертигации из бака Б*)
	 tTimerValue_poliv_with_fert	: TIME:=t#60m;  (* Ограничение полива с фертигацией *)
	 tTimerValue_poliv_finish	: TIME:=t#3s;  (*Пауза перед статусом завршения полива для обновления регистров *)

	Timer_valve				: TON;
	Timer_valveQ			: BOOL;
	 tTimerValue_valve_water	: TIME:=t#60m;  (* Максимальное время открытия клапана подачи воды в теплицу*)

	TRIG_start_poliv			:	R_TRIG;
	TRIG_valve_tank_F		:	F_TRIG;
	TRIG_valve_tank_R		:	R_TRIG;

	TRIG_level_tank_low		:	R_TRIG;
	TRIG_level_tank_high		:	R_TRIG;

	Timer_light_avg			: TON;
	 tTimer_light_avg			: TIME:=t#1m;
	Timer_light_avgQ			: BOOL;
	Bool_poliv_before_fert		: 	BOOL;

	TRIG_poliv_break			:	R_TRIG;


	FertA_liters				:	REAL;
	FertB_liters				:	REAL;
	gisterezis_lux				:	INT:=1000;
(*	Poliv_before_fert			:	INT:=0; *)
	Timer_poliv_with_fertQ		: 	BOOL;


	max_EC					:	REAL;
	pi_fertA2 			: FB_CTRL_PI;
	pi_fertB2 			: FB_CTRL_PI;

	set_kf_fert		: INT:=12;
	start_cfg_pi_par	:BOOL;
	setA, setB, actA, actB, fOutA, fOutB	:REAL;

	avg_light_ma			: FB_CTRL_MOVING_AVERAGE;
	stParams_avg_light	: ST_CTRL_MOVING_AVERAGE_PARAMS;


	start_cfg_avg_light			:BOOL;

	avg_light					: REAL;
	arr_table					: ARRAY[1..20] OF FLOAT;
	Cnt_water_pipe			:UDINT;
	pwm_data_A	: REAL;
	pwm_cnt_A	: UDINT;
	pwm_avg_A	: REAL;
	pwm_data_B	: REAL;
	pwm_cnt_B	: UDINT;
	pwm_avg_B	: REAL;
	tank_level_low	:BOOL;
	tank_level_high	:BOOL;

END_VAR
IF NOT start_cfg_avg_light THEN

	stParams_avg_light.tCtrlCycleTime			:= T#60s;
	stParams_avg_light.tTaskCycleTime 			:= T#10ms;
	stParams_avg_light.nSamplesToFilter		:= 20;
	stParams_avg_light.pWorkArray_ADR		:= ADR(arr_table);
	stParams_avg_light.nWorkArray_SIZEOF		:= SIZEOF(arr_table);
	start_cfg_avg_light							:= TRUE;
END_IF

avg_light_ma(fIn:=Modbus.Teplica_light_lux, fManSyncValue :=0, bSync:=0, eMode:=eCTRL_MODE_ACTIVE,bHold:=0, stParams:=stParams_avg_light,  fOut =>avg_light);
Modbus.Teplica_avg_lux	:=	avg_light;


start_cfg_pi_par:=	FALSE;
IF NOT start_cfg_pi_par THEN


	pi_par_fertA.bARWOnIPartOnly:=0;
	pi_par_fertA.fKp:=300000*0.7;
	pi_par_fertA.fOutMaxLimit:=32765*0.7;
	pi_par_fertA.fOutMinLimit:=32765*0.25;

(*	pi_par_fertA.fOutMinLimit:=16800; *)
(*	pi_par_fertA.fOutMinLimit:=13100; *)
(*	pi_par_fertA.fOutMinLimit:=11460; *)
	pi_par_fertA.tCtrlCycleTime:=T#4s;
	pi_par_fertA.tTaskCycleTime:=T#10ms;
	pi_par_fertA.tTn:=T#8s;

	pi_par_fertB.bARWOnIPartOnly:=0;
	pi_par_fertB.fKp:=300000*0.7;
	pi_par_fertB.fOutMaxLimit:=32765*0.7;
	pi_par_fertB.fOutMinLimit:=32765*0.25;
(*	pi_par_fertB.fOutMinLimit:=16800; *)
(*	pi_par_fertB.fOutMinLimit:=13100; *)
(*	pi_par_fertA.fOutMinLimit:=11460; *)
	pi_par_fertB.tCtrlCycleTime:=T#4s;
	pi_par_fertB.tTaskCycleTime:=T#10ms;
	pi_par_fertB.tTn:=T#8s;

	start_cfg_pi_par			:=	TRUE;

END_IF


IF (Kf_calc_fertA = 0) THEN
	Kf_calc_fertA := 48;
END_IF
IF (Kf_calc_fertB = 0) THEN
	Kf_calc_fertB := 48;
END_IF
IF (Modbus.Teplica_fert_kf = 0) THEN
	Modbus.Teplica_fert_kf := 48;
END_IF

CASE Modbus.Teplica_fert_kf OF

64:
		pi_par_fertA.fOutMaxLimit:=32765*0.4;
		pi_par_fertA.fOutMinLimit:=32765*0.3;
		pi_par_fertB.fOutMaxLimit:=32765*0.5;
		pi_par_fertB.fOutMinLimit:=32765*0.4;

48:
		pi_par_fertA.fOutMaxLimit:=32765*0.45;
		pi_par_fertA.fOutMinLimit:=32765*0.35;
		pi_par_fertB.fOutMaxLimit:=32765*0.55;
		pi_par_fertB.fOutMinLimit:=32765*0.45;


32:
		pi_par_fertA.fOutMaxLimit:=32765*0.6;
		pi_par_fertA.fOutMinLimit:=32765*0.45;
		pi_par_fertB.fOutMaxLimit:=32765*0.7;
		pi_par_fertB.fOutMinLimit:=32765*0.5;


END_CASE


setA		:=	1/INT_TO_REAL(Modbus.Teplica_fert_kf);

setB		:=	1/INT_TO_REAL(Modbus.Teplica_fert_kf);


(*
Trigger_water_impulse_teplica(CLK:=HW_impulse_water_teplica);
Trigger_fertA_impulse_teplica(CLK:=HW_impulse_fertA_teplica);
Trigger_fertB_impulse_teplica(CLK:=HW_impulse_fertB_teplica);

IF Trigger_water_impulse_teplica.Q THEN
	Modbus.Teplica_impulse_water_cnt	:= 	Modbus.Teplica_impulse_water_cnt+1;
END_IF


IF Trigger_fertA_impulse_teplica.Q THEN
	Modbus.Teplica_impulse_fertA_cnt	:= 	Modbus.Teplica_impulse_fertA_cnt+1;
END_IF
IF Trigger_fertB_impulse_teplica.Q THEN
	Modbus.Teplica_impulse_fertB_cnt	:= 	Modbus.Teplica_impulse_fertB_cnt+1;
END_IF
*)
tTimerValue_poliv_all	:=	UDINT_TO_TIME(60*1000*Modbus.Teplica_set_max_poliv_time);
tTimerValue_1_clear	:=	UDINT_TO_TIME(60*1000*Modbus.Teplica_set_clear_time);
tTimerValue_2_fertA	:=	UDINT_TO_TIME(60*1000*Modbus.Teplica_set_max_fertA_time);
tTimerValue_3_clear	:=	UDINT_TO_TIME(60*1000*Modbus.Teplica_set_finish_clear_time);
tTimerValue_4_fertB	:=	UDINT_TO_TIME(60*1000*Modbus.Teplica_set_max_fertB_time);

Timer_poliv_all();
Timer_poliv_with_fert();
Timer_1_clear();
Timer_2_fertA();
Timer_3_clear();
Timer_4_fertB();
Timer_valve();
Timer_poliv_finish();
Timer_calc_kf();

TRIG_start_poliv(CLK :=Modbus.Teplica_poliv_active);
TRIG_poliv_break(CLK :=Modbus.Teplica_poliv_break);

TRIG_valve_tank_F(CLK:=HW_water_tank_teplica_level);
TRIG_valve_tank_R(CLK:=HW_water_tank_teplica_level);

IF (Modbus.Teplica_tank_level <1000) THEN
	tank_level_low	:=	TRUE;
	tank_level_high	:=	FALSE;
END_IF
IF (Modbus.Teplica_tank_level >1200) THEN
	tank_level_high	:=	TRUE;
	tank_level_low	:=	FALSE;
END_IF



TRIG_level_tank_low(CLK:= tank_level_low);
TRIG_level_tank_high(CLK:= tank_level_high);

Modbus.Teplica_tank_teplica_level	:=	HW_water_tank_teplica_level;

IF (TRIG_valve_tank_F.Q OR TRIG_level_tank_low.Q ) THEN
	Timer_valve(IN:=NOT Timer_valveQ , PT:=tTimerValue_valve_water , Q=>Timer_valveQ , ET=> );
	HW_valve_pomp_teplica :=	TRUE;
	Modbus.Teplica_valve_water_in		:=	TRUE;
END_IF


IF (TRIG_valve_tank_R.Q	OR Timer_valveQ = TRUE OR TRIG_level_tank_high.Q) THEN
	HW_valve_pomp_teplica :=	FALSE;
	Modbus.Teplica_valve_water_in		:=	FALSE;
	Timer_valveQ	:= FALSE;
	Timer_valve.IN	:= FALSE;
END_IF



IF (TRIG_start_poliv.Q  AND Modbus.Teplica_tank_level > 400 )   THEN
		pwm_data_A	:=	0;
		pwm_cnt_A	:=	0;
		pwm_avg_A	:=	0;
		pwm_data_B	:=	0;
		pwm_cnt_B	:=	0;
		pwm_avg_B	:=	0;


		Cnt_water_pipe	:=	0;
		Poliv_liters	:=	0;
		FertA_liters	:=	0;
		FertB_liters	:=	0;
		Cnt_water_fertA_start	:=	0;
		Cnt_water_fertB_start	:=	0;
		Cnt_water_finish_clear	:=	0;
		Cnt_water_finish_clear_start		:=	0;
		Modbus.Teplica_impulse_water_cnt	:=	0;
		Modbus.Teplica_impulse_fertA_cnt	:=	0;
		Modbus.Teplica_impulse_fertB_cnt	:=	0;
		Modbus.Teplica_cnt_water_pipe			:=	0;

		Modbus.Teplica_time_elapsed_poliv :=0;
		Modbus.Teplica_time_elapsed_fertA :=0;
		Modbus.Teplica_time_elapsed_fertB :=0;
		max_EC	:=	0;
		Timer_1_clearQ			:= FALSE;
		Timer_2_fertAQ			:= FALSE;
		Timer_3_clearQ			:= FALSE;
		Timer_4_fertBQ			:= FALSE;
		Timer_poliv_finishQ		:= FALSE;
		Timer_calc_kfQ			:=FALSE;
		Bool_poliv_before_fert		:=FALSE;
		Modbus.Teplica_pomp_poliv:=TRUE;

		Timer_poliv_all.IN := FALSE;
		Timer_poliv_with_fert.IN := FALSE;
		Timer_1_clear.IN := FALSE;
		Timer_2_fertA.IN:=FALSE;
		Timer_3_clear.IN := FALSE;
		Timer_4_fertB.IN:=FALSE;
		Timer_calc_kf.IN	:=	FALSE;
		Timer_poliv_finish.IN := FALSE;

		 t_Started_poliv := TIME();
		Timer_poliv_all(IN:=NOT Timer_poliv_allQ , PT:=tTimerValue_poliv_all , Q=>Timer_poliv_allQ , ET=> );
		Timer_poliv_with_fert(IN:=NOT Timer_poliv_with_fertQ , PT:=tTimerValue_poliv_with_fert , Q=>Timer_poliv_with_fertQ , ET=> );
		Timer_1_clear(IN:=NOT Timer_1_clearQ , PT:=tTimerValue_1_clear , Q=>Timer_1_clearQ , ET=> );
		Modbus.Teplica_poliv_status_PLC:=2;
		IF  (Modbus.Teplica_zone_poliv = 0) THEN
			Modbus.Teplica_poliv_message_PLC:=1;
		ELSE
			Modbus.Teplica_poliv_message_PLC:=2;
		END_IF


END_IF

IF (Modbus.Teplica_poliv_status_PLC=2  ) THEN
	Cnt_water_pipe	:=	Modbus.Teplica_cnt_water_pipe;
	Poliv_liters 	:= 	UDINT_TO_REAL(Modbus.Teplica_impulse_water_cnt)/INT_TO_REAL(Modbus.Teplica_poliv_kf);
	FertA_liters	:=	UDINT_TO_REAL(Modbus.Teplica_impulse_fertA_cnt)/INT_TO_REAL(Modbus.Teplica_fertA_kf);
	FertB_liters	:=	UDINT_TO_REAL(Modbus.Teplica_impulse_fertB_cnt)/INT_TO_REAL(Modbus.Teplica_fertB_kf);
	Modbus.Teplica_time_elapsed_poliv :=(TIME_TO_UDINT( TIME() - t_Started_poliv))/1000;

(*	pi_fertA2(fSetpointValue:=setA, fActualValue := actA, fManSyncValue :=0, bSync:=0, eMode:=2,bHold:=0, stParams:=pi_par_fertA, fOut => );
	pi_fertB2(fSetpointValue:=setB, fActualValue :=actB, fManSyncValue :=0, bSync:=0, eMode:=2,bHold:=0, stParams:=pi_par_fertB, fOut => );
	fOutA	:=	pi_fertA2.fOut;
	fOutB	:=	pi_fertB2.fOut;
*)

	IF (Modbus.Teplica_sensor_soil_EC > max_EC) THEN
		max_EC	:=	Modbus.Teplica_sensor_soil_EC;
	END_IF

(* промывка и фертигация   OR Modbus.Teplica_set_poliv_before_fert >Poliv_liters*)

	IF (Modbus.Teplica_type_poliv = TRUE) THEN  (* Полив с фертигацией*)
		IF (NOT Timer_1_clear.Q AND Bool_poliv_before_fert	= FALSE)  THEN
			IF (Modbus.Teplica_type_fert = FALSE) THEN
				IF  (Modbus.Teplica_zone_poliv = 0) THEN
						Modbus.Teplica_poliv_message_PLC:=3;
				ELSE
						Modbus.Teplica_poliv_message_PLC:=4;
				END_IF

			ELSE
				IF  (Modbus.Teplica_zone_poliv = 0) THEN
					Modbus.Teplica_poliv_message_PLC:=5;
				ELSE
					Modbus.Teplica_poliv_message_PLC:=6;
				END_IF

			END_IF
		END_IF


		IF ((Timer_1_clear.Q OR Poliv_liters>Modbus.Teplica_set_poliv_before_fert) AND Bool_poliv_before_fert=FALSE) THEN

			Timer_1_clear.IN 		:= FALSE;
			Bool_poliv_before_fert	:= TRUE;
			IF (Modbus.Teplica_type_fert = FALSE) THEN
				 (*Fert A *)
				IF  (Modbus.Teplica_zone_poliv = 0) THEN
					Modbus.Teplica_poliv_message_PLC:=7;
				ELSE
					Modbus.Teplica_poliv_message_PLC:=8;
				END_IF

				Modbus.Teplica_pomp_fertA :=  TRUE;  (*включение насоса фертигации из бака А*)
				Timer_2_fertA(IN:=NOT Timer_2_fertAQ , PT:=tTimerValue_2_fertA , Q=>Timer_2_fertAQ , ET=> );
				t_Started_fertA := TIME();
				Cnt_water_fertA_start :=Modbus.Teplica_impulse_water_cnt;
				Cnt_water_calc_kf_start	:=Poliv_liters;
				Cnt_fertA_calc_kf_start:=FertA_liters;

			ELSE
				 (*Fert B *)
				IF  (Modbus.Teplica_zone_poliv = 0) THEN
					Modbus.Teplica_poliv_message_PLC:=9;
				ELSE
					Modbus.Teplica_poliv_message_PLC:=10;
				END_IF

				Modbus.Teplica_pomp_fertB :=  TRUE;   (*включение насоса фертигации из бака B*)
				Timer_4_fertB(IN:=NOT Timer_4_fertBQ , PT:=tTimerValue_4_fertB , Q=>Timer_4_fertBQ , ET=> );
				t_Started_fertB := TIME();
				Cnt_water_fertB_start :=Modbus.Teplica_impulse_water_cnt;
				Cnt_water_calc_kf_start	:=Poliv_liters;
				Cnt_fertB_calc_kf_start:=FertB_liters;

			END_IF
		END_IF
		IF ( (Timer_2_fertA.Q OR FertA_liters > Modbus.Teplica_set_fertA) AND Modbus.Teplica_pomp_fertA =  TRUE) THEN
			 (*start finish clear *)
			IF  (Modbus.Teplica_zone_poliv = 0) THEN
				Modbus.Teplica_poliv_message_PLC:=11;
			ELSE
				Modbus.Teplica_poliv_message_PLC:=12;
			END_IF

			Modbus.Teplica_pomp_fertA :=  FALSE; (*отключение насоса фертигации из бака А*)
			Modbus.Teplica_time_elapsed_fertA :=(TIME_TO_UDINT( TIME() - t_Started_fertA))/1000;
			Modbus.Cnt_water_fertA	:=	Modbus.Teplica_impulse_water_cnt -Cnt_water_fertA_start;
			Timer_2_fertA.IN:=FALSE;
			Cnt_water_finish_clear_start		:=	Modbus.Teplica_impulse_water_cnt;
			Timer_3_clear(IN:=NOT Timer_3_clearQ , PT:=tTimerValue_3_clear , Q=>Timer_3_clearQ , ET=> );
		END_IF
		IF ( (Timer_4_fertB.Q OR FertB_liters > Modbus.Teplica_set_fertB) AND Modbus.Teplica_pomp_fertB =  TRUE ) THEN
			 (*start finish clear *)
			IF  (Modbus.Teplica_zone_poliv = 0) THEN
				Modbus.Teplica_poliv_message_PLC:=13;
			ELSE
				Modbus.Teplica_poliv_message_PLC:=14;
			END_IF

			Modbus.Teplica_pomp_fertB :=  FALSE; (*отключение насоса фертигации из бака B*)
			Modbus.Teplica_time_elapsed_fertB :=(TIME_TO_UDINT( TIME() - t_Started_fertB))/1000;
			Modbus.Cnt_water_fertB	:=	Modbus.Teplica_impulse_water_cnt -Cnt_water_fertB_start;

			Timer_4_fertB.IN:=FALSE;
			Cnt_water_finish_clear_start		:=	Modbus.Teplica_impulse_water_cnt;
			Timer_3_clear(IN:=NOT Timer_3_clearQ , PT:=tTimerValue_3_clear , Q=>Timer_3_clearQ , ET=> );
		END_IF

		IF  (Modbus.Teplica_pomp_fertA =  TRUE) THEN
			actA		:=	1/Kf_calc_fertA;
			pi_fertA2(fSetpointValue:=setA, fActualValue := actA, fManSyncValue :=0, bSync:=0, eMode:=2,bHold:=0, stParams:=pi_par_fertA, fOut => );
			fOutA	:=	pi_fertA2.fOut;
			Modbus.Teplica_time_elapsed_fertA :=(TIME_TO_UDINT( TIME() - t_Started_fertA))/1000;
			Modbus.Cnt_water_fertA	:=	Modbus.Teplica_impulse_water_cnt -Cnt_water_fertA_start;
			Timer_calc_kf(IN:=NOT Timer_calc_kfQ , PT:=t#4s , Q=>Timer_calc_kfQ , ET=> );
			IF (Timer_calc_kf.Q)	THEN
				vol_water	:=	Poliv_liters-Cnt_water_calc_kf_start;
				vol_fertA		:=	FertA_liters-Cnt_fertA_calc_kf_start;
				IF (vol_fertA > 0 ) THEN
					Kf_calc_fertA	:= 	 vol_water/vol_fertA;
				ELSE
					Kf_calc_fertA	:=	1000;
				END_IF
				Cnt_water_calc_kf_start	:=Poliv_liters;
				Cnt_fertA_calc_kf_start:=FertA_liters;
				Timer_calc_kfQ	:=	FALSE;
				Timer_calc_kf.IN	:=	FALSE;
			END_IF
			fert_pwm_levelA	:=	 REAL_TO_UINT(fOutA);
(*			IF (vol_fertA>0.05 ) THEN *)
				pwm_data_A		:=	pwm_data_A + fert_pwm_levelA;
				pwm_cnt_A		:=	pwm_cnt_A + 1;
				pwm_avg_A		:=	pwm_data_A / pwm_cnt_A;
(*			END_IF *)
		ELSE
			fert_pwm_levelA	:=	0;

		END_IF



		IF (Modbus.Teplica_pomp_fertB =  TRUE) THEN
			actB		:=	1/Kf_calc_fertB;
			pi_fertB2(fSetpointValue:=setB, fActualValue :=actB, fManSyncValue :=0, bSync:=0, eMode:=2,bHold:=0, stParams:=pi_par_fertB, fOut => );
			fOutB	:=	pi_fertB2.fOut;
			Modbus.Teplica_time_elapsed_fertB :=(TIME_TO_UDINT( TIME() - t_Started_fertB))/1000;
			Modbus.Cnt_water_fertB	:=	Modbus.Teplica_impulse_water_cnt -Cnt_water_fertB_start;
			Timer_calc_kf(IN:=NOT Timer_calc_kfQ , PT:=t#4s , Q=>Timer_calc_kfQ , ET=> );
			IF (Timer_calc_kf.Q)	THEN
				vol_water	:=	Poliv_liters-Cnt_water_calc_kf_start;
				vol_fertB		:=	FertB_liters-Cnt_fertB_calc_kf_start;
				IF (vol_fertB > 0 ) THEN
					Kf_calc_fertB	:= 	 vol_water/vol_fertB;
				ELSE
					Kf_calc_fertB	:=	1000;
				END_IF

				Cnt_water_calc_kf_start	:=Poliv_liters;
				Cnt_fertB_calc_kf_start:=FertB_liters;
				Timer_calc_kfQ	:=	FALSE;
				Timer_calc_kf.IN	:=	FALSE;
			END_IF
			fert_pwm_levelB	:=	 REAL_TO_UINT(fOutB);
(*			IF (vol_fertB>0.05 ) THEN *)
				pwm_data_B		:=	pwm_data_B + fert_pwm_levelB;
				pwm_cnt_B		:=	pwm_cnt_B + 1;
				pwm_avg_B		:=	pwm_data_B / pwm_cnt_B;
(*			END_IF *)
		ELSE
			fert_pwm_levelB	:=	0;

		END_IF


		IF (Modbus.Teplica_poliv_message_PLC =11 OR Modbus.Teplica_poliv_message_PLC = 12 OR Modbus.Teplica_poliv_message_PLC = 13  OR Modbus.Teplica_poliv_message_PLC = 14) THEN
			Cnt_water_finish_clear	:=	UDINT_TO_REAL(Modbus.Teplica_impulse_water_cnt-Cnt_water_finish_clear_start)/Modbus.Teplica_poliv_kf;
		END_IF


		IF (Timer_poliv_with_fert.Q=TRUE OR   Modbus.Teplica_poliv_break=TRUE OR Timer_3_clear.Q=TRUE OR Cnt_water_finish_clear > Modbus.Teplica_set_finish_clear_vol  )THEN


			Modbus.Teplica_max_EC		:=	max_EC;

			Modbus.Teplica_poliv_active:= FALSE;
			Modbus.Teplica_pomp_poliv:=FALSE;
			Modbus.Teplica_pomp_fertA :=  FALSE;
			Modbus.Teplica_pomp_fertB :=  FALSE;
			Timer_poliv_all.IN := FALSE;
			Timer_poliv_with_fert.IN := FALSE;
			Timer_1_clear.IN := FALSE;
			Timer_2_fertA.IN:=FALSE;
			Timer_3_clear.IN := FALSE;
			Timer_4_fertB.IN:=FALSE;
			Timer_calc_kf.IN	:=	FALSE;
			Timer_1_clearQ			:= FALSE;
			Timer_2_fertAQ			:= FALSE;
			Timer_3_clearQ			:= FALSE;
			Timer_4_fertBQ			:= FALSE;

			IF (Modbus.Teplica_type_fert = FALSE) THEN
				 (*finished poliv with fert A*)
				IF  (Modbus.Teplica_zone_poliv = 0) THEN
					Modbus.Teplica_poliv_message_PLC:=15;
				ELSE
					Modbus.Teplica_poliv_message_PLC:=16;
				END_IF

			ELSE
				IF  (Modbus.Teplica_zone_poliv = 0) THEN
					Modbus.Teplica_poliv_message_PLC:=17;
				ELSE
					Modbus.Teplica_poliv_message_PLC:=18;
				END_IF

			END_IF

			Modbus.Teplica_poliv_status_PLC :=  10;
			Timer_poliv_finish(IN:=NOT Timer_poliv_finishQ, PT:=tTimerValue_poliv_finish , Q=>Timer_poliv_finishQ , ET=> );
		END_IF
		ELSE
			fert_pwm_levelA:=0;
			fert_pwm_levelB:=0;
	END_IF

	IF (Modbus.Teplica_type_poliv = FALSE) THEN (*Полив без фертигации*)
		IF (Timer_poliv_all.Q=TRUE OR (Poliv_liters > Modbus.Teplica_set_poliv)  OR Modbus.Teplica_poliv_break=TRUE   )THEN
			(*finished only poliv *)
			IF  (Modbus.Teplica_zone_poliv = 0) THEN
					Modbus.Teplica_poliv_message_PLC:=19;
			ELSE
					Modbus.Teplica_poliv_message_PLC:=20;
			END_IF

			Modbus.Teplica_poliv_active:= FALSE;
			Modbus.Teplica_pomp_poliv:=FALSE;
			Modbus.Teplica_pomp_fertA :=  FALSE;
			Modbus.Teplica_pomp_fertB :=  FALSE;
			Timer_poliv_all.IN := FALSE;
			Timer_poliv_with_fert.IN := FALSE;
			Timer_1_clear.IN := FALSE;
			Timer_2_fertA.IN:=FALSE;
			Timer_3_clear.IN := FALSE;
			Timer_4_fertB.IN:=FALSE;
			Timer_1_clearQ			:= FALSE;
			Timer_2_fertAQ			:= FALSE;
			Timer_3_clearQ			:= FALSE;
			Timer_4_fertBQ			:= FALSE;
			Modbus.Teplica_poliv_status_PLC :=  10;
		END_IF
	END_IF
	ELSE
		fert_pwm_levelA:=0;
		fert_pwm_levelB:=0;
END_IF

Modbus.Teplica_fert_actA			:=	Kf_calc_fertA;
Modbus.Teplica_fert_actB			:=	Kf_calc_fertB;
Modbus.Teplica_fert_pwm_levelA	:=	REAL_TO_INT(100*fert_pwm_levelA/32765);
Modbus.Teplica_fert_pwm_levelB	:=	REAL_TO_INT(100*fert_pwm_levelB/32765);
Modbus.Teplica_pwm_avg_A		:=	REAL_TO_INT(100*pwm_avg_A/32765);
Modbus.Teplica_pwm_avg_B		:=	REAL_TO_INT(100*pwm_avg_B/32765);









(*LIGHT TEPLICA *)

IF (Modbus.Teplica_light = FALSE) THEN

(*	IF ((Modbus.Teplica_avg_lux > Modbus.Teplica_light_set_low+gisterezis_lux OR Modbus.Teplica_temp_air>25) OR Modbus.Teplica_light_allow = FALSE  ) THEN
		Modbus.Teplica_light :=FALSE;
		HW_teplica_light		:=	FALSE;
	END_IF
*)
	IF ((Modbus.Teplica_avg_lux <  Modbus.Teplica_light_set_low-gisterezis_lux  AND Modbus.Teplica_temp_air<27) AND Modbus.Teplica_light_allow ) THEN
		Modbus.Teplica_light:=TRUE;
		HW_teplica_light		:=	TRUE;
	END_IF

END_IF

IF (Modbus.Teplica_light = TRUE) THEN

	IF ((Modbus.Teplica_avg_lux  >  Modbus.Teplica_light_set_low+gisterezis_lux  OR Modbus.Teplica_temp_air>28) OR Modbus.Teplica_light_allow = FALSE  ) THEN
		Modbus.Teplica_light :=FALSE;
		HW_teplica_light		:=	FALSE;
	END_IF

(*	IF ((Modbus.Teplica_avg_lux <  Modbus.Teplica_light_set_low-gisterezis_lux ) AND Modbus.Teplica_light_allow ) THEN
		Modbus.Teplica_light:=TRUE;
		HW_teplica_light		:=	TRUE;
	END_IF
*)

END_IF



(*HEAT TEPLICA *)

	IF ((Modbus.Teplica_temp_air > Modbus.Teplica_temp_set_low+1) ) THEN
		Modbus.Teplica_heat :=FALSE;
		HW_teplica_heat		:= FALSE;
	END_IF

	IF ((Modbus.Teplica_temp_air <  Modbus.Teplica_temp_set_low-1 ) ) THEN
		Modbus.Teplica_heat:=TRUE;
		HW_teplica_heat		:=	TRUE;
	END_IF


(*HEAT TANK TEPLICA *)

	IF ((Modbus.Teplica_temp_water_tank > Modbus.Teplica_set_temp_tank+1)  OR HW_teplica_heat = TRUE   OR Modbus.Teplica_tank_level < 400 ) THEN
		Modbus.Teplica_tank_heat :=FALSE;
		HW_teplica_tank_heat		:= FALSE;
	END_IF

	IF ((Modbus.Teplica_temp_water_tank <  Modbus.Teplica_set_temp_tank-1 ) AND HW_teplica_heat = FALSE   AND Modbus.Teplica_tank_level > 400) THEN
		Modbus.Teplica_tank_heat:=TRUE;
		HW_teplica_tank_heat		:=	TRUE;
	END_IF




(*VENT  TEPLICA *)

	IF ((Modbus.Teplica_temp_air < Modbus.Teplica_temp_set_high-1)   ) THEN
		Modbus.Teplica_vent			 :=FALSE;
		HW_teplica_vent				:=FALSE;
	END_IF

	IF ((Modbus.Teplica_temp_air >  Modbus.Teplica_temp_set_high+1 ) ) THEN
		Modbus.Teplica_vent	:=TRUE;
		HW_teplica_vent		:=TRUE;
	END_IF


	IF (Modbus.Teplica_temp_air < Modbus.Teplica_set_temp_window_open-1 ) THEN
		HW_teplica_window_opener		:=FALSE;
		Modbus.Teplica_window_opener	:=FALSE;
	END_IF
	IF (Modbus.Teplica_temp_air >  Modbus.Teplica_set_temp_window_open+1 AND   Modbus.Street_temp > 0 ) THEN
		HW_teplica_window_opener		:=TRUE;
		Modbus.Teplica_window_opener	:=TRUE;
	END_IF


	IF (Modbus.Teplica_temp_air < Modbus.Teplica_set_temp_pomp_cold-1   ) THEN
		HW_teplica_pomp_cold		:=FALSE;
		Modbus.Teplica_pomp_cold	:=FALSE;
	END_IF
	IF (Modbus.Teplica_temp_air >  Modbus.Teplica_set_temp_pomp_cold+1 AND   Modbus.Street_temp >10 ) THEN
		HW_teplica_pomp_cold		:=TRUE;
		Modbus.Teplica_pomp_cold	:=TRUE;
	END_IF
END_PROGRAM

(* POU FB_GreenhouseWindowControl, ST *)
FUNCTION_BLOCK FB_GreenhouseWindowControl
VAR
    state            : INT := 0;
    target_level     : UINT := 0;
    active_target    : UINT := 0;
    current_level_int: UINT := 0;
    move_timer       : TON;
    start_closing    : BOOL := FALSE;
    start_opening    : BOOL := FALSE;
    close_cond       : BOOL;
    open60_cond      : BOOL;
    open30_cond      : BOOL;
END_VAR

VAR_INPUT
    Street_temp                    : REAL;
    Parnik_set_temp_street_min     : REAL;
    Parnik_air_temp                : REAL;
    Parnik_set_auto_window         : BOOL;
    Parnik_manual_level_window     : UINT;
    Parnik_temp_step1_window       : UINT;
    Parnik_temp_step2_window       : UINT;
END_VAR

VAR_OUTPUT
    HW_power_supply_parnik  : BOOL;
    HW_power_polarity_parnik: BOOL;
    Parnik_current_level_window : UINT;
END_VAR
(* --- Вычисление целевого уровня --- *)
IF Parnik_set_auto_window THEN
    close_cond  := (Parnik_air_temp < (UINT_TO_REAL(Parnik_temp_step1_window) - 2.0))
                   OR (Street_temp < Parnik_set_temp_street_min);
    open60_cond := (Parnik_air_temp > (UINT_TO_REAL(Parnik_temp_step2_window) + 2.0))
                   AND (Street_temp > Parnik_set_temp_street_min);
    open30_cond := (Parnik_air_temp > (UINT_TO_REAL(Parnik_temp_step1_window) + 2.0))
                   AND (Parnik_air_temp < UINT_TO_REAL(Parnik_temp_step2_window))
                   AND (Street_temp > Parnik_set_temp_street_min);
    IF close_cond THEN
        target_level := 0;
    ELSIF open60_cond THEN
        target_level := 2;
    ELSIF open30_cond THEN
        target_level := 1;
    ELSE
        target_level := current_level_int;
    END_IF
ELSE
    target_level := Parnik_manual_level_window;
END_IF

(* --- Конечный автомат --- *)
CASE state OF
    0: (* IDLE *)
        IF target_level <> current_level_int THEN
            active_target := target_level;
            IF (current_level_int = 0) AND (active_target > 0) THEN
                start_opening := TRUE;
                state := 2;
            ELSE
                start_closing := TRUE;
                state := 1;
            END_IF
        END_IF

    1: (* CLOSING *)
        IF start_closing THEN
            move_timer.PT := T#60S;
            move_timer.IN := TRUE;
            start_closing := FALSE;
        ELSE
            move_timer.IN := TRUE;
        END_IF
        move_timer(); (* ВАЖНО: вызов таймера *)
        IF move_timer.Q THEN
            move_timer.IN := FALSE;
            current_level_int := 0;
            state := 0;
        END_IF

    2: (* OPENING *)
        IF start_opening THEN
            CASE active_target OF
                1: move_timer.PT := T#15S;
                2: move_timer.PT := T#30S;
                3: move_timer.PT := T#50S;
            ELSE
                move_timer.PT := T#0S;
            END_CASE
            move_timer.IN := TRUE;
            start_opening := FALSE;
        ELSE
            move_timer.IN := TRUE;
        END_IF
        move_timer(); (* ВАЖНО: вызов таймера *)
        IF move_timer.Q THEN
            move_timer.IN := FALSE;
            current_level_int := active_target;
            state := 0;
        END_IF
END_CASE

(* --- Выходы двигателя --- *)
IF state = 1 THEN
    HW_power_supply_parnik   := TRUE;
    HW_power_polarity_parnik := FALSE; (* закрытие *)
ELSIF state = 2 THEN
    HW_power_supply_parnik   := TRUE;
    HW_power_polarity_parnik := TRUE;  (* открытие *)
ELSE
    HW_power_supply_parnik   := FALSE;
    HW_power_polarity_parnik := FALSE;
END_IF

Parnik_current_level_window := current_level_int;
END_FUNCTION_BLOCK

(* POU FB_Mqtt_Subscribe_V10, ST *)
(* @NESTEDCOMMENTS := 'Yes' *)
(* @PATH := '\/_Generic\/Mqtt' *)
(* @OBJECTFLAGS := '0, 8' *)
(* @SYMFILEFLAGS := '2048' *)
FUNCTION_BLOCK FB_Mqtt_Subscribe_V10
VAR_INPUT
	sTopic	: STRING[255];
	bAccept	: BOOL := FALSE; (* When false, subscribe but do not set bNewValue output *)
END_VAR
VAR_OUTPUT
	sValue		: STRING[255];
	bNewValue	: BOOL := FALSE;
	bBusy		: BOOL := FALSE;
END_VAR
VAR_IN_OUT
	stMqttSettings	: ST_MqttSettings;
END_VAR
VAR
	iState 				: INT := 0;
	bSubscribeSent		: BOOL := FALSE;
	bSubAckReceived		: BOOL := FALSE;
	iTopicLength		: INT := 0;
	wTopicLength		: WORD;
	stMqttTelegram		: ST_MqttTelegram;
	fbMqttEncodeLength	: FB_Mqtt_EncodeLength_V10;
	bLength1			: BYTE;
	bLength2			: BYTE;
	bLength3			: BYTE;
	bLength4			: BYTE;
	bLengthAmount		: BYTE;

	wPackageIdentifier			: WORD;
	wTelegramPackageIdentifier	: WORD;
END_VAR
VAR CONSTANT
	C_STARTUP			: INT := 0;
	C_BUILD_TELEGRAM	: INT := 100;
	C_SEND_WAIT			: INT := 110;
	C_CHECK_TELEGRAM	: INT := 200;
	C_IDLE				: INT := 500;
END_VAR

(* @END_DECLARATION := '0' *)
CASE iState OF
	C_STARTUP:
		wPackageIdentifier 	:= 0;
		bSubscribeSent		:= FALSE;
		bSubAckReceived		:= FALSE;
		bNewValue			:= FALSE;
		sValue 				:= '';
		bBusy				:= FALSE;

		IF stMqttSettings.bValidConnection THEN
			iState := C_IDLE;
		END_IF;

	(* build publish telegram *)
	C_BUILD_TELEGRAM:
		bBusy 								:= TRUE;
		wPackageIdentifier 					:= stMqttSettings.wPackageIdentifier;
		stMqttSettings.wPackageIdentifier 	:= stMqttSettings.wPackageIdentifier + 1;
		iTopicLength						:= LEN(sTopic);

		FC_Mqtt_ClearTelegram_V10(
			stMqttTelegram	:= stMqttTelegram,
			stMqttSettings	:= stMqttSettings
		);

		wTopicLength := iTopicLength;
		wTopicLength := HOST_TO_BE16(wTopicLength);

		wTelegramPackageIdentifier := HOST_TO_BE16(wPackageIdentifier);

		(* Calculate length *)
		(* 2 byte package identifier, 2 byte length topic, x byte length topic, 1 byte QoS *)
		fbMqttEncodeLength(
			dwLength := 2 + 2 + iTopicLength + 1,
			bLength1 => bLength1,
			bLength2 => bLength2,
			bLength3 => bLength3,
			bLength4 => bLength4,
			bAmount	 => bLengthAmount
		);

		(* MQTT Control Packet type *)
		stMqttTelegram.arMqttData[0] := 130;

		(* Remaining Length *)
		CASE bLengthAmount OF
			1:
				stMqttTelegram.arMqttData[1] := bLength1;

			2:
				stMqttTelegram.arMqttData[1] := bLength1;
				stMqttTelegram.arMqttData[2] := bLength2;

			3:
				stMqttTelegram.arMqttData[1] := bLength1;
				stMqttTelegram.arMqttData[2] := bLength2;
				stMqttTelegram.arMqttData[3] := bLength3;

			4:
				stMqttTelegram.arMqttData[1] := bLength1;
				stMqttTelegram.arMqttData[2] := bLength2;
				stMqttTelegram.arMqttData[3] := bLength3;
				stMqttTelegram.arMqttData[4] := bLength4;

			ELSE
				iState 					:= C_STARTUP;
				stMqttSettings.bError	:= TRUE;
		END_CASE;

		(* Packet Identifier MSB *)
		stMqttTelegram.arMqttData[1 + bLengthAmount] := WORD_TO_BYTE(wTelegramPackageIdentifier);
		(* Packet Identifier LSB *)
		stMqttTelegram.arMqttData[2 + bLengthAmount] := WORD_TO_BYTE(SHR(wTelegramPackageIdentifier, 8));
		(* Length MSB Topic *)
		stMqttTelegram.arMqttData[3 + bLengthAmount] := WORD_TO_BYTE(wTopicLength);
		(* Length MSB Topic *)
		stMqttTelegram.arMqttData[4 + bLengthAmount] := WORD_TO_BYTE(SHR(wTopicLength, 8));

		(* Add topic *)
		MEMCPY(
			destAddr	:= ADR(stMqttTelegram.arMqttData[5 + bLengthAmount]),
		    srcAddr		:= ADR(sTopic),
			n  			:= iTopicLength
		);

		(* 1 byte header, x byte variable length, 2 byte package identifier, 2 byte topic lenght, x byte topic, 1 byte QoS *)
		stMqttTelegram.nDataLength := 1 + bLengthAmount + 2 + 2 + iTopicLength + 1;

		iState := C_SEND_WAIT;

	(* send telegram *)
	C_SEND_WAIT:
		IF stMqttSettings.stMqttSendTelegram.nDataLength = 0 THEN
			FC_Mqtt_CopyTelegram_V10(
				stMqttSrcTelegram	:= stMqttTelegram,
				stMqttDestTelegram	:= stMqttSettings.stMqttSendTelegram,
				stMqttSettings		:= stMqttSettings
			);

			bSubscribeSent	:= TRUE;
			iState			:= C_IDLE;
		END_IF;

		IF NOT stMqttSettings.bValidConnection THEN
			iState := C_STARTUP;
		END_IF;

	(* check telegram *)
	C_CHECK_TELEGRAM:
		bBusy 			:= TRUE;

		IF
			stMqttSettings.stMqttReceivedPublishTelegram.bHasData
			AND stMqttSettings.stMqttReceivedPublishTelegram.sTopic = sTopic
		THEN
			FC_Mqtt_ClearTelegram_V10(
				stMqttTelegram	:= stMqttSettings.stMqttReceivedTelegram,
				stMqttSettings	:= stMqttSettings
			);
			stMqttSettings.stMqttReceivedPublishTelegram.bHasData := FALSE;

			sValue		:= stMqttSettings.stMqttReceivedPublishTelegram.sValue;
			bNewValue 	:= TRUE;
		END_IF;

		iState := C_IDLE;

	(* idle *)
	C_IDLE:
		bBusy 		:= FALSE;
		bNewValue	:= FALSE;

		IF
			stMqttSettings.bValidConnection
			AND NOT bSubscribeSent
			AND NOT bSubAckReceived
		THEN
			iState := C_BUILD_TELEGRAM;
		END_IF;

		(* Check for correct SubAck *)
		IF
			bSubscribeSent
			AND stMqttSettings.stMqttReceivedTelegram.nDataLength = 5
			AND stMqttSettings.stMqttReceivedTelegram.arMqttData[0] = 144
			AND stMqttSettings.stMqttReceivedTelegram.arMqttData[1] = 3
			AND stMqttSettings.stMqttReceivedTelegram.arMqttData[2] = WORD_TO_BYTE(wTelegramPackageIdentifier)
			AND stMqttSettings.stMqttReceivedTelegram.arMqttData[3] = WORD_TO_BYTE(SHR(wTelegramPackageIdentifier, 8))
			AND stMqttSettings.stMqttReceivedTelegram.arMqttData[4] = 0
		THEN
			FC_Mqtt_ClearTelegram_V10(
				stMqttTelegram	:= stMqttSettings.stMqttReceivedTelegram,
				stMqttSettings	:= stMqttSettings
			);
			bSubAckReceived := TRUE;
		END_IF;

		(* Check for error SubAck *)
		IF
			bSubscribeSent
			AND stMqttSettings.stMqttReceivedTelegram.nDataLength = 5
			AND stMqttSettings.stMqttReceivedTelegram.arMqttData[0] = 144
			AND stMqttSettings.stMqttReceivedTelegram.arMqttData[1] = 3
			AND stMqttSettings.stMqttReceivedTelegram.arMqttData[2] = WORD_TO_BYTE(wTelegramPackageIdentifier)
			AND stMqttSettings.stMqttReceivedTelegram.arMqttData[3] = WORD_TO_BYTE(SHR(wTelegramPackageIdentifier, 8))
			AND stMqttSettings.stMqttReceivedTelegram.arMqttData[4].7 = 1
		THEN
			stMqttSettings.bError := TRUE;
		END_IF;

		(* Check for publish *)
		IF
			bSubAckReceived
			AND stMqttSettings.stMqttReceivedPublishTelegram.bHasData
			AND bAccept
		THEN
			iState := C_CHECK_TELEGRAM;
		END_IF;

		IF NOT stMqttSettings.bValidConnection THEN
			iState := C_STARTUP;
		END_IF;

	ELSE
		iState := C_STARTUP;
END_CASE

(*	END_FUNCTION_BLOCK	*)
END_FUNCTION_BLOCK
